TYPE M3TranslationGotoProcedureStatuses :
STRUCT
	///Is the M3GotoProcedure in a busy state?
	busyStatus: BusyStatus;
	///Is the M3GotoProcedure in a healthy state?
	healthStatus: HealthStatus;
END_STRUCT
END_TYPE

(* stored: Version 1.1.0.1, ProductVersion 3.1.4019.2
   DUT M3TranslationGotoProcedureStatuses: Id {c225cd10-a45b-48ee-b413-56fff71ef47c} *)
